# B&R Automation Studio project Lab1
Automation Studio 4.5.2.102; Default project

## Configuration Simulation

CPU , AutomationRuntime M4.01, Build 4.1.2, Vc V3.96.7

### Task classes (Cpu.sw)
```
Cyclic#1 (cycle 10000 us):
  Program1 <- Program1.prg
Libraries: AsIecCon, astime, MtrCtrl
```

### Hardware
```
PLC1 : PC_any v1.1.0.0 (OrderNumber=PC)
  VolatileGlobalPvSize = 4096
  PreserveNonVolatileSystemSettings = 0
  XLinkUseDefault = 0
  Cyclic1Duration = 10000
```

## Logical view

Binary libraries used (declarations not repeated): Runtime, OPERATOR, AsIecCon, astime

### Package Logical/Libraries - Global libraries

### Library Logical/Libraries/MtrCtrl (ANSIC) - A new source library

#### MtrCtrl.fun - Exported functions and function blocks
```iecst
(********************************************************************
 * COPYRIGHT --
 ********************************************************************
 * Library: MtrCtrl
 * File: MtrCtrl.fun
 * Author: admin
 * Created: October 16, 2018
 ********************************************************************
 * Functions and function blocks of library MtrCtrl
 ********************************************************************)

FUNCTION_BLOCK FB_Motor (*TODO: Add your comment here*)
	VAR_INPUT
		U : REAL;
	END_VAR
	VAR_OUTPUT
		W : REAL;
		Phi : REAL;
	END_VAR
	VAR
		Tm : REAL;
		Ke : REAL;
		Dt : REAL;
		Integrator : FB_Integrator;
	END_VAR
END_FUNCTION_BLOCK

FUNCTION_BLOCK FB_Integrator (*TODO: Add your comment here*)
	VAR_INPUT
		In : REAL;
	END_VAR
	VAR_OUTPUT
		Out : REAL;
	END_VAR
	VAR
		Dt : REAL;
	END_VAR
END_FUNCTION_BLOCK

FUNCTION_BLOCK FB_Controller (*TODO: Add your comment here*)
	VAR_INPUT
		E : REAL;
	END_VAR
	VAR_OUTPUT
		U : REAL;
	END_VAR
	VAR
		k_p : REAL;
		k_i : REAL;
		Integrator : FB_Integrator;
		iyOld : REAL;
		max_abs_value : REAL;
		Dt : REAL;
		abs_in_1 : REAL;
		abs_out_1 : REAL;
		abs_in_2 : REAL;
	END_VAR
END_FUNCTION_BLOCK
```

#### FB_Integrator.c
```c
/********************************************************************
 * COPYRIGHT --
 ********************************************************************
 * Library: MtrCtrl
 * File: FB_Integrator.c
 * Author: admin
 * Created: October 16, 2018
 ********************************************************************
 * Implementation of library MtrCtrl
 ********************************************************************/

#include <bur/plctypes.h>
#ifdef __cplusplus
	extern "C"
	{
#endif

	#include "MtrCtrl.h"

#ifdef __cplusplus
	};
#endif

/* TODO: Add your comment here */
void FB_Integrator(struct FB_Integrator* inst)
{
	inst->out+=inst->in;
}
```

#### FB_Motor.c
```c
/********************************************************************
 * COPYRIGHT --
 ********************************************************************
 * Library: MtrCtrl
 * File: FB_Motor.c
 * Author: admin
 * Created: October 16, 2018
 ********************************************************************
 * Implementation of library MtrCtrl
 ********************************************************************/

#include <bur/plctypes.h>
#ifdef __cplusplus
	extern "C"
	{
#endif

	#include "MtrCtrl.h"

#ifdef __cplusplus
	};
#endif

/* TODO: Add your comment here */
void FB_Motor(struct FB_Motor* inst)
{
	inst->integrator.in=(inst->u/inst->Ke-inst->w)*inst->dt/inst->Tm; inst->integrator.out=inst->w;
	FB_Integrator(&(inst->integrator)); inst->w=inst->integrator.out;
	inst->integrator.in=inst->w*inst->dt; inst->integrator.out=inst->phi; FB_Integrator(&(inst->integrator)); inst->phi=inst->integrator.out;
}
```

#### FB_Regulator.c
```c
/********************************************************************
 * COPYRIGHT --
 ********************************************************************
 * Library: MtrCtrl
 * File: FB_Controller.c
 * Author: admin
 * Created: October 16, 2018
 ********************************************************************
 * Implementation of library MtrCtrl
 ********************************************************************/

#include <bur/plctypes.h>
#ifdef __cplusplus
	extern "C"
	{
#endif

	#include "MtrCtrl.h"

#ifdef __cplusplus
	};
#endif

/* TODO: Add your comment here */
void FB_Regulator(struct FB_Regulator* inst)
{
	inst->integrator.in=inst->e * inst->k_i * inst->dt + inst->iyOld; FB_Integrator(&(inst->integrator)); inst->e_kp=inst->e*inst->k_p;
	inst->e_kp=(inst->e_kp > inst->max_abs_value || inst->e_kp < - inst->max_abs_value)?((inst->e_kp>0)?inst-
		>max_abs_value:-inst->max_abs_value):inst->e_kp; inst->e_kp+=inst->integrator.out;
	inst->u=(inst->e_kp > inst->max_abs_value || inst->e_kp < - inst->max_abs_value)?((inst->e_kp>0)?inst-
		>max_abs_value:-inst->max_abs_value):inst->e_kp; inst->iyOld=inst->u-inst->e_kp;
}
```

### Program Logical/Program1 (ANSIC) - A new program

#### Program.c - Implementation code
```c
/********************************************************************
 * COPYRIGHT --
 ********************************************************************
 * Program: Program1
 * File: Program1.c
 * Author: admin
 * Created: October 16, 2018
 ********************************************************************
 * Implementation of program Program1
 ********************************************************************/

#include <bur/plctypes.h>

#ifdef _DEFAULT_INCLUDES
	#include <AsDefault.h>
#endif

void _INIT ProgramInit(void)
{
	fb_motor.dt=0.01;
	fb_motor.Ke=2;
	fb_motor.Tm=0.4;
	fb_motor.integrator.dt=0.01;

	fb_motor2.dt=0.01;
	fb_motor2.Ke=2;
	fb_motor2.Tm=0.4;
	fb_motor2.integrator.dt=0.01;

	fb_regulator.dt=0.01;
	fb_regulator.k_p=8;
	fb_regulator.k_i=20;
	fb_regulator.max_abs_value=24;
	fb_regulator.integrator.dt=0.01;

	enable=1; count=0;
}
void _CYCLIC ProgramCyclic(void)
{
	if(enable)
	{
		count+=10;
		if(count<=2500)
		{

			speed=0;

		}
		else
		{
			speed=6;
			if(count>=5000)
			{

				count=0;
			}
		}
	}
	fb_regulator.e=speed - fb_motor.w;
	fb_motor2.u=speed;
	FB_Regulator(&fb_regulator);
	fb_motor.u=fb_regulator.u;
	FB_Motor(&fb_motor);
	FB_Motor(&fb_motor2);
}
```

#### Program.var - Local variables
```iecst
(********************************************************************
 * COPYRIGHT --
 ********************************************************************
 * Program: Program1
 * File: Program1.var
 * Author: admin
 * Created: October 16, 2018
 ********************************************************************
 * Local variables of program Program1
 ********************************************************************)
VAR
	fb_controller : FB_Controller := (0);
	fb_motor : FB_Motor := (0);
	fb_motor2 : FB_Motor := (0);
	speed : REAL := 0.0;
	enable : BOOL := FALSE;
	count : INT := 0;
END_VAR
```
